FUNCTION_BLOCK MotorFailureReport_FB
VAR_INPUT
	AxisCtrlPtr			: POINTER TO Basic_axis_typ ;
	StationID 			: eStationNo;
	
	(*Ref_ev_MOTOR_POSITION   : REFERENCE TO ev_MOTOR_POSITION_ERROR REF= ev_MOTOR_POSITION_ERROR;
	Ref_ev_MOTOR_Speed      : REFERENCE TO ev_MOTOR_SPEED_ERROR    REF= ev_MOTOR_SPEED_ERROR;	
	Ref_ev_HOME_NOT_FOUND   : REFERENCE TO ev_MOTOR_HOME_NOT_FOUND REF= ev_MOTOR_HOME_NOT_FOUND;
	Ref_ev_OVER_CURRENT     : REFERENCE TO ev_MOTOR_OVER_CURRENT   REF= ev_MOTOR_OVER_CURRENT;

	Ref_ev_MOTOR_OVER_TEMP      : REFERENCE TO  ev_MOTOR_OVER_TEMP        REF= ev_MOTOR_OVER_TEMP;
	Ref_ev_MOTOR_FEEDBACK_ERROR : REFERENCE TO	ev_MOTOR_FEEDBACK_ERROR   REF=  ev_MOTOR_FEEDBACK_ERROR ;
	Ref_ev_MOTOR_GENERAL_ERROR 	: REFERENCE TO	ev_MOTOR_GENERAL_ERROR    REF=  ev_MOTOR_GENERAL_ERROR ;
	Ref_ev_MOTOR_STALLED		: REFERENCE TO  ev_MOTOR_STALLED          REF=  ev_MOTOR_STALLED;
	Ref_ev_MOTOR_SUPPLY_ERROR 	: REFERENCE TO	ev_MOTOR_SUPPLY_ERROR     REF=  ev_MOTOR_SUPPLY_ERROR ;
 	Ref_ev_PLC_ILLEGAL_MSG  	: REFERENCE TO	ev_PLC_ILLEGAL_MSG        REF= 	ev_PLC_ILLEGAL_MSG  ;
	Ref_ev_PLC_ILLEGAL_PARAM 	: REFERENCE TO	ev_PLC_ILLEGAL_PARAM      REF= 	ev_PLC_ILLEGAL_PARAM ;
	Ref_ev_Drive_Not_Enabled 	: REFERENCE TO  ev_MOTOR_DRIVE_NOT_ENABLED REF= 	ev_MOTOR_DRIVE_NOT_ENABLED ;
	
	Ref_ev_DRIVE_NOT_READY    	: REFERENCE TO	ev_MOTOR_DRIVE_NOT_READY  REF= 	ev_MOTOR_DRIVE_NOT_READY ;
	Ref_ev_Drive_ComError		: REFERENCE TO  ev_MOTOR_DRIVE_COM_ERROR  REF= 	ev_MOTOR_DRIVE_COM_ERROR ;
	Ref_ev_BRAKE_RESISTOR_ERROR : REFERENCE TO  ev_BRAKE_RESISTOR_ERROR   REF= 	ev_BRAKE_RESISTOR_ERROR ;
	*)
	

                                                                            
	                                                                        


	
	
END_VAR
VAR
	LastErrorId			: UDINT;
	PrevErrorId			: UDINT;
	AxisLastErrorCount  : UDINT := 0;
	Pop_Delay	 		: TON;
	ErrorID_Delay 		: TON;
	lastEventID: enumMotorEvents;
	MotorErrorQ			: Queue;
	QErrorCounter       : UDINT;
	//
	LogMsgInit          : BOOL := TRUE;
	LogMsg_0 			: LogMsg ;
	//Get old events from Q
	PrevMotorEvents		: Eh_ErrorEntry_typ;
	ThreadName		    : STRING[20];	
	fbPrgmBasic			:FB_PrgmBasic;
	
	//EventParameters:EventParam_Typ;	
	//EventHeader:EventHeader_Typ;	
	
END_VAR

//Classifier
//Method






IF AxisCtrlPtr <> 0 THEN
		
	IF LogMsgInit THEN      
		LogMsgInit := FALSE ;
		ThreadName := AxisCtrlPtr^.Input.Parameter.ThreadName;
		CONCAT(  ThreadName,'Re');
		fnLogMsgInit(ADR(LogMsg_0), ThreadName, ADR(LogGlobalArray), ADR(CONST_ZERO));
		LogMsg_0.Enable:= 		TRUE;
	END_IF

	IF AxisCtrlPtr^.Output.Error.ErrorCount > 0 AND AxisCtrlPtr^.Input.Command.ErrorAcknowledge = FALSE THEN
		ErrorID_Delay.PT := T#25MS ;	
		Pop_Delay.IN := TRUE;	
			
			
	END_IF
	
	
	IF Pop_Delay.Q THEN
		Pop_Delay.IN := FALSE;
		AxisCtrlPtr^.Input.Command.ErrorAcknowledge := TRUE;
	END_IF	
	Pop_Delay();
	
	//Add code for clear error	
	ErrorID_Delay.IN := AxisCtrlPtr^.Output.Error.ErrorCount  = 0 AND AxisCtrlPtr^.Output.Status.FAULT ;
	ErrorID_Delay.PT := T#100MS ;
	ErrorID_Delay();
						
	IF ErrorID_Delay.Q THEN
		
		AxisCtrlPtr^.Input.Command.ClearFault := TRUE;
		
	END_IF
	

	//Check if there is new error
	IF AxisCtrlPtr^.Output.Error.fbErrorHandler.EntriesCount <> 0 AND
	  lastEventID<> AxisCtrlPtr^.Output.Error.ErrorEntry.MotorEvents AND 
	  AxisCtrlPtr^.Output.Error.ErrorEntry.MotorEvents <> enumMotorEvents.NoEvents THEN		
		
		AxisLastErrorCount := AxisCtrlPtr^.Output.Error.fbErrorHandler.EntriesCount;
	 	
		IF Meth_GetEvent( AxisCtrlPtr^.Output.Error.ErrorEntry ) = FALSE THEN
			
			MotorErrorQ.Enqueue(ADR(AxisCtrlPtr^.Output.Error.ErrorEntry),SIZEOF(Eh_ErrorEntry_typ));	
			IF AxisCtrlPtr^.Input.Parameter.pFlowID <> 0 THEN
			   fnLogMsg(ADR(LogMsg_0), LOG_INFO, 'Event is locked keep msg in Q Send Event ID %d,ErrorId =%d, flowid %d',
								AxisCtrlPtr^.Output.Error.ErrorEntry.MotorEvents  ,
								UDINT_TO_DINT(AxisCtrlPtr^.Output.Error.ErrorEntry.ErrorId),							
								AxisCtrlPtr^.Input.Parameter.pFlowID^);
			ELSE
				
			   fnLogMsg(ADR(LogMsg_0), LOG_INFO, 'Event is locked keep msg in Q Send Event ID %d,ErrorId =%d THERE IS NO LINK TO FLOW ID:',
								AxisCtrlPtr^.Output.Error.ErrorEntry.MotorEvents  ,
								UDINT_TO_DINT(AxisCtrlPtr^.Output.Error.ErrorEntry.ErrorId),							
								0);
			END_IF							
		ELSE

							
			IF AxisCtrlPtr^.Output.Error.ErrorEntry.ErrorId <>0 THEN
				
				LastErrorId := 	AxisCtrlPtr^.Output.Error.ErrorEntry.ErrorId;	
				
			END_IF
			
			PrevErrorId := AxisCtrlPtr^.Output.Error.ErrorEntry.ErrorId;
	
		END_IF
		
		lastEventID := 	AxisCtrlPtr^.Output.Error.ErrorEntry.MotorEvents;
		
	ELSIF MotorErrorQ.CheckQReadAvailable() THEN
					
	
			IF MotorErrorQ.ReadCurrentEntry(ADR(PrevMotorEvents),SIZEOF(Eh_ErrorEntry_typ)) THEN	
	
				IF Meth_GetEvent( PrevMotorEvents )  THEN
						
					MotorErrorQ.Dequeue(ADR(PrevMotorEvents),SIZEOF(PrevMotorEvents));
					
					fnLogMsg(ADR(LogMsg_0), LOG_INFO, 'Dequeue Event ID %d,ErrorId =%d',
								PrevMotorEvents.MotorEvents  ,
								UDINT_TO_DINT(PrevMotorEvents.ErrorId),							
								0);
	
				END_IF
			END_IF
	END_IF
	
END_IF
//fnLogTransfer FUNCTION call
fbPrgmBasic();

fnLogTransfer(ADR(LogMsg_0));

METHOD Meth_GetEvent : BOOL
VAR_INPUT
	ErrorEntry		: Eh_ErrorEntry_typ;
END_VAR
VAR
	EventSentOk:  	BOOL;
END_VAR
   EventSentOk := FALSE;

	CASE ErrorEntry.MotorEvents OF
		enumMotorEvents.NoEvents				:
			 EventSentOk := TRUE;//No Event	
		enumMotorEvents.MotorPositionError      :
			
			IF Meth_SendEvent( Ref_ev_MOTOR_POSITION ) = FALSE THEN
				EventSentOk := FALSE;
			ELSE
				EventSentOk := TRUE;
			END_IF
				
		enumMotorEvents.MotorSpeedError	        :
			IF Meth_SendEvent(  Ref_ev_MOTOR_Speed ) = FALSE THEN
				EventSentOk := FALSE;
			ELSE
				EventSentOk := TRUE;
			END_IF
		enumMotorEvents.MotorHomeNotFound	    :
			IF Meth_SendEvent( Ref_ev_HOME_NOT_FOUND ) = FALSE THEN
				EventSentOk := FALSE;
			ELSE
				EventSentOk := TRUE;
			END_IF
		enumMotorEvents.MotorOverCurrent	    :
			IF Meth_SendEvent( Ref_ev_OVER_CURRENT ) = FALSE THEN
				EventSentOk := FALSE;
			ELSE
				EventSentOk := TRUE;
			END_IF
		enumMotorEvents.MotorOverTemp		    :
			IF Meth_SendEvent(Ref_ev_MOTOR_OVER_TEMP ) = FALSE THEN
				EventSentOk := FALSE;
			ELSE
				EventSentOk := TRUE;
			END_IF
		enumMotorEvents.MotorFeedBackErr	    :
			IF Meth_SendEvent( Ref_ev_MOTOR_FEEDBACK_ERROR ) = FALSE THEN
				EventSentOk := FALSE;
			ELSE
				EventSentOk := TRUE;
			END_IF
		enumMotorEvents.MotorGeneralError		:
			IF Meth_SendEvent(Ref_ev_MOTOR_GENERAL_ERROR ) = FALSE THEN
				EventSentOk := FALSE;
			ELSE
				EventSentOk := TRUE;
			END_IF
		enumMotorEvents.MotorStalled			:
			IF Meth_SendEvent( Ref_ev_MOTOR_STALLED ) = FALSE THEN
				EventSentOk := FALSE;
			ELSE
				EventSentOk := TRUE;
			END_IF
		enumMotorEvents.MotorSupplyError		:
			IF Meth_SendEvent( Ref_ev_MOTOR_SUPPLY_ERROR ) = FALSE THEN
				EventSentOk := FALSE;
			ELSE
				EventSentOk := TRUE;
			END_IF
		enumMotorEvents.PLCillegalMsg			:
			IF Meth_SendEvent(Ref_ev_PLC_ILLEGAL_MSG ) = FALSE THEN
				EventSentOk := FALSE;
			ELSE
				EventSentOk := TRUE;
			END_IF
		enumMotorEvents.PLCIllegalParam			:
			IF Meth_SendEvent( Ref_ev_PLC_ILLEGAL_PARAM ) = FALSE THEN
				EventSentOk := FALSE;
			ELSE
				EventSentOk := TRUE;
			END_IF
		enumMotorEvents.DriveNotEnabled		    :
			IF Meth_SendEvent(Ref_ev_Drive_Not_Enabled ) = FALSE THEN
				EventSentOk := FALSE;
			ELSE
				EventSentOk := TRUE;
			END_IF
		enumMotorEvents.DriveNotReady           :
			IF Meth_SendEvent(Ref_ev_DRIVE_NOT_READY  ) = FALSE THEN
				EventSentOk := FALSE;
			ELSE
				EventSentOk := TRUE;
			END_IF
		enumMotorEvents.DriveComError           :
			IF Meth_SendEvent(Ref_ev_Drive_ComError ) = FALSE THEN
				EventSentOk := FALSE;
			ELSE
				EventSentOk := TRUE;
			END_IF
		enumMotorEvents.BreakResistorError:
			IF Meth_SendEvent( Ref_ev_BRAKE_RESISTOR_ERROR)= FALSE THEN
				EventSentOk := FALSE;
			ELSE
				EventSentOk := TRUE;
			END_IF
		
	END_CASE
	
		IF EventSentOk  AND ErrorEntry.MotorEvents <> enumMotorEvents.NoEvents THEN
			IF AxisCtrlPtr^.Input.Parameter.pFlowID <> 0 THEN
				fnLogMsg(ADR(LogMsg_0), LOG_INFO, 'Send Event ID %d,ErrorId =%d, FlowId=%d',
					AxisCtrlPtr^.Output.Error.ErrorEntry.MotorEvents  ,
					UDINT_TO_DINT(AxisCtrlPtr^.Output.Error.ErrorEntry.ErrorId),							
					AxisCtrlPtr^.Input.Parameter.pFlowID^);
			ELSE
				fnLogMsg(ADR(LogMsg_0), LOG_INFO, 'Send Event ID %d,ErrorId =%d, THERE IS NO LINK TO FLOWID',
					AxisCtrlPtr^.Output.Error.ErrorEntry.MotorEvents  ,
					UDINT_TO_DINT(AxisCtrlPtr^.Output.Error.ErrorEntry.ErrorId),							
					0);
		
			END_IF		
		END_IF

	Meth_GetEvent := EventSentOk;
END_METHOD

METHOD Meth_SendEvent : BOOL
VAR_INPUT
	RefEvent : REFERENCE TO EventHelper;
END_VAR
VAR

	Dummy :DINT :=0;
//	pFlowID :POINTER TO DINT;
END_VAR
IF __ISVALIDREF(RefEvent) THEN
		
		EventHeader.SubsysID :=			 AxisCtrlPtr^.Input.Parameter.SubsysID; 
		IF AxisCtrlPtr^.Input.Parameter.pFlowID <> 0 THEN
			EventHeader.pFlowID :=  AxisCtrlPtr^.Input.Parameter.pFlowID;					 // Flow ID
		ELSE
			EventHeader.pFlowID :=  ADR(Dummy);
		END_IF	
		EventParameters.MotorID := 		 AxisCtrlPtr^.Input.Parameter.MotorID; 	// Motor ID
		EventParameters.VendorNameID :=  AxisCtrlPtr^.Input.Parameter.Drive.VendorNameID;	// Vendor name ID

		fbPrgmBasic.mEventThrow(RefEvent,ADR(EventHeader),ADR(EventParameters) );			//RefEvent();
		Meth_SendEvent := TRUE;

END_IF
END_METHOD

END_FUNCTION_BLOCK

(* stored: Version 1.1.0.1, ProductVersion 3.1.4024.3
   POU MotorFailureReport_FB: Id {20eea4f0-96bf-0356-09b1-09cafda83e4c}, SpecialFunc None
   Method Meth_GetEvent: Id {ca711a49-4463-08c1-0a73-929709d939e4}
   Method Meth_SendEvent: Id {17a229e8-5c5e-0243-0858-7f4311c71782} *)
